Universal Robots PolyScope program: MAIN_bak20230705.urp

Program MAIN_bak20230705 (installation=GD directory=/programs/GD createdIn=5.13.0 lastSavedIn=5.13.0 robotSerialNumber=20205000017)
Calibrated DH parameters: a=[-0.000157, -0.56303, -0.236706, -0.000074, -0.000109, 0]; d=[0.181705, 47.632387, 369.599619, -417.058513, 0.119878, 0.115667]; alpha=[1.570881, -0.005074, -0.001247, 1.56886, -1.570997, 0]; deltaTheta=[0, -0.405485, 5.544791, 1.143886, -0.000009, -0.000001]
InitVariablesNode
BeforeStart
  Script file /programs/GD/ROVI/ROVI_RESET.script
    | def ROVI_RESET():
    |   if (not socket_open(host,port,socket_name)):
    |     rovi_err=902
    |     return False
    |   end
    |   socket_send_line("X0()",socket_name)
    |   ret=socket_read_line(socket_name,socket_timeout)
    |   if (ret == "OK"):
    |     rovi_err=0
    |   elif (ret == "NG"):
    |     rovi_err=to_num(socket_read_line(socket_name,socket_timeout))
    |   else:
    |     ret="NG"
    |     rovi_err=903
    |   end
    |   socket_close(socket_name)
    |   if (rovi_err != 0):
    |     if (is_popup):
    |       popup(str_cat(ret,rovi_err),title="X0",warning=True,blocking=True)
    |     end
    |     return False
    |   else:
    |     return True
    |   end
    | end
  Script file /programs/GD/ROVI/ROVI_CAPTURE.script
    | def ROVI_CAPTURE():
    |   Y1=[0.0,0.0,0.0,0.0]
    | #  p=get_actual_tool_flange_pose()
    |   p=Bucket
    |   if (not socket_open(host,port,socket_name)):
    |     rovi_err=902
    |     return False
    |   end
    |   socket_send_string("X1(",socket_name)
    |   socket_send_string(p[0],socket_name)
    |   socket_send_string(",",socket_name)
    |   socket_send_string(p[1],socket_name)
    |   socket_send_string(",",socket_name)
    |   socket_send_string(p[2],socket_name)
    |   socket_send_string(",",socket_name)
    |   socket_send_string(p[3],socket_name)
    |   socket_send_string(",",socket_name)
    |   socket_send_string(p[4],socket_name)
    |   socket_send_string(",",socket_name)
    |   socket_send_string(p[5],socket_name)
    |   socket_send_line(")",socket_name)
    |   ret=socket_read_line(socket_name,socket_timeout)
    |   if (ret == "OK"):
    |     rovi_err=0
    |     f=socket_read_ascii_float(4,socket_name,socket_timeout)
    |     while (f[0]!=4):
    |       sleep(0.3)
    |       f=socket_read_ascii_float(4,socket_name,socket_timeout)
    |     end
    |     i=0
    |     while (i<4):
    |       Y1[i]=f[i+1]
    |       i=i+1
    |     end
    |   elif (ret == "NG"):
    |     rovi_err=to_num(socket_read_line(socket_name,socket_timeout))
    |   else:
    |     ret="NG"
    |     rovi_err=903
    |   end
    |   socket_close(socket_name)
    |   if (rovi_err != 0):
    |     if (is_popup):
    |       popup(str_cat(ret,rovi_err),title="X1",warning=True,blocking=True)
    |     end
    |     return False
    |   else:
    |     return True
    |   end
    | end
  Script file /programs/GD/ROVI/ROVI_SOLVE.script
    | def ROVI_SOLVE(is_popup=is_popup):
    |   buf=p[10000.0,0.0,0.0,0.0,0.0,0.0]
    |   if (not socket_open(host,port,socket_name)):
    |     rovi_err=902
    |     return False
    |   end
    |   socket_send_line("X2()",socket_name)
    |   ret=socket_read_line(socket_name,socket_timeout)
    |   if (ret == "OK"):
    |     rovi_err=0
    |     f=socket_read_ascii_float(6,socket_name,socket_timeout)
    |     while (f[0]!=6):
    |       sleep(0.3)
    |       f=socket_read_ascii_float(6,socket_name,socket_timeout)
    |     end
    |     counter=0
    |     while (counter<6):
    |       buf[counter]=f[counter+1]
    |       counter=counter+1
    |     end
    |   elif (ret == "NG"):
    |     rovi_err=to_num(socket_read_line(socket_name,socket_timeout))
    |   else:
    |     ret="NG"
    |     rovi_err=903
    |   end
    |   sleep(1.0)
    |   socket_close(socket_name)
    |   if (rovi_err != 0):
    |     if (is_popup):
    |       popup(str_cat(ret,rovi_err),title="X2",warning=True,blocking=True)
    |     end
    |   end
    |   return buf
    | end
  Script file /programs/GD/ROVI/ROVI_RECIPE.script
    | def ROVI_RECIPE(recipe):
    |   if (not socket_open(host,port,socket_name)):
    |     rovi_err=902
    |     return False
    |   end
    |   socket_send_line(str_cat(str_cat("X3(",recipe),")"),socket_name)
    |   ret=socket_read_line(socket_name,socket_timeout)
    |   if (ret == "OK"):
    |     rovi_err=0
    |   elif (ret == "NG"):
    |     rovi_err=to_num(socket_read_line(socket_name,socket_timeout))
    |   else:
    |     ret="NG"
    |     rovi_err=903
    |   end
    |   socket_close(socket_name)
    |   if (rovi_err != 0):
    |     if (is_popup):
    |       popup(str_cat(ret,rovi_err),title="X3",warning=True,blocking=True)
    |     end
    |     return False
    |   else:
    |     return True
    |   end
    | end
  Script file /programs/GD/ROVI/ROVI_PARAM.script
    | def ROVI_PARAM(prm_name,prm_value=None):
    |   Y8=0.0
    |   if (not socket_open(host,port,socket_name)):
    |     rovi_err=902
    |     return False
    |   end
    |   socket_send_string("X8(",socket_name)
    |   socket_send_string(prm_name,socket_name)
    |   if (prm_value != None):
    |     socket_send_string(" ",socket_name)
    |     socket_send_string(prm_value,socket_name)
    |   end
    |   socket_send_line(")",socket_name)
    |   ret=socket_read_line(socket_name,socket_timeout)
    |   if (ret == "OK"):
    |     rovi_err=0
    |     if (prm_value == None):  # rosparam get
    |       Y8=to_num(socket_read_line(socket_name,socket_timeout))
    |     else:    # rosparam set
    |       f=1
    |     end
    |   elif (ret == "NG"):
    |     rovi_err=to_num(socket_read_line(socket_name,socket_timeout))
    |   else:
    |     ret="NG"
    |     rovi_err=903
    |   end
    |   socket_close(socket_name)
    |   if (rovi_err != 0):
    |     if (is_popup):
    |       popup(str_cat(ret,rovi_err),title="X8",warning=True,blocking=True)
    |     end
    |     return False
    |   else:
    |     return True
    |   end
    | end
  Script file /programs/GD/CONTROL/STATUS_CONTROL.script
    | def CHECK_VT_STATUS():
    |   write_output_boolean_register(8, read_input_boolean_register(64))   # GPBO_PCOK
    |   write_output_boolean_register(9, read_input_boolean_register(65))   # GPBO_YCAMOK
    |   write_output_integer_register(5, read_input_integer_register(24))   # GPIO_PayloadNo
    | end
  Script file /programs/GD/CONTROL/CYCLE_CONTROL.script
    | def GET_REG(prg_no):
    |   WorkPosNo=read_input_integer_register(4)-1                       # GPII_WorkPosNo
    |   CaptIndex[WorkPosNo]=read_input_integer_register(21)-1           # GPII_CaptColNo
    |   CaptRowNo=read_input_integer_register(20)-1        # GPII_CaptRowNo
    |   CaptStepZ=read_input_integer_register(6) / 1000.0         # GPII_CaptStepZ
    |   ReCaptNo=0
    |   if (prg_no==1203):
    |     ReCaptNo=read_input_integer_register(22)                # GPII_ReCaptNo
    |   end
    |   ReCaptZ=read_input_integer_register(7) / 1000.0         # GPII_ReCaptZ
    |   CutOffZDef=read_input_integer_register(11) / 1000.0          # GPII_CutOffZ
    |   CrankDepthFull=read_input_integer_register(10) / 1000.0   # GPII_FullDepth
    | end
    | 
    | def POSE_SUB(p, teach_frame):
    |   return pose_trans(inv(teach_frame), p)
    | end
    | 
    | def GET_BUCKET_UPPER(pos=0):
    |   if UseNewCaptPos:
    |     p=POSE_SUB(CaptPoint_C, BucketM)
    |     pX=[BKWidth/2,CaptPointL_dX,BKWidth-CaptPointR_dX]
    |     p[0]=pX[pos]
    |   else:
    |     captpos=[CaptPoint_C,CaptPoint_L,CaptPoint_R]
    |     p=captpos[pos]
    |     p=POSE_SUB(p, BucketM)
    |   end
    |   return p
    | end
    | 
    | def SET_BUCKET_DEF():
    |   BucketM=pBucketM
    |   if (WorkPosNo<0):
    |     Bucket=pBucketC
    |   else:
    |     Bucket=pBucket[WorkPosNo]
    |   end
    | end
    | 
    | def SET_BUCKET():
    |   SET_BUCKET_DEF()
    |   Bucket[2]=Bucket[2]-CaptStepZ*CaptRowNo
    | end
    | 
    | def SET_CV():
    |   CV=pCV
    | end
    | 
    | def SET_CAPT_INDEX():
    |   CaptIndexWk=CaptIndex[WorkPosNo]
    |   ReCaptZWk=0
    |   if (prg_no==1203):
    |     if   (ReCaptNo==0):
    |       if (CaptIndexWk==0):
    |         if (0<=DistPillarBak):
    |           CaptIndexWk=1
    |         else:
    |           CaptIndexWk=2
    |         end
    |         ReCaptZWk=0
    |       else:
    |         CaptIndexWk=0
    |         ReCaptZWk=0
    |       end
    |     elif (ReCaptNo==1):
    |       if (CaptIndexWk==0):
    |         CaptIndexWk=0
    |         ReCaptZWk=-ReCaptZ
    |       else:
    |         CaptIndexWk=CaptIndexWk
    |         ReCaptZWk=-ReCaptZ
    |       end
    |     else:
    |       if (CaptIndexWk==0):
    |         CaptIndexWk=0
    |         ReCaptZWk=ReCaptZ
    |       else:
    |         CaptIndexWk=CaptIndexWk
    |         ReCaptZWk=ReCaptZ
    |       end
    |     end
    |   end
    | end
    | 
    | def GET_CAPTPOS():
    |   SET_BUCKET()
    |   SET_CAPT_INDEX()
    |   if UseNewCaptPos:
    |     p=GET_BUCKET_UPPER(CaptIndexWk)
    |     p[2]=p[2]-ReCaptZWk
    |   else:
    |     captpos=[CaptPoint_C,CaptPoint_L,CaptPoint_R]
    |     p=captpos[CaptIndexWk]
    |     p[2]=p[2]-ReCaptZWk
    |     p=POSE_SUB(p, BucketM)
    |   end
    |   return p
    | end
    | 
    | def CHECK_CAPTPOS():
    |   isOK=((CaptStepZ*(read_input_integer_register(20)-1)) < (read_input_integer_register(9) / 1000.0))
    |   return isOK
    | end
    | 
    | def GET_ZSLIDE_POS(p):
    |   p[2]=p[2]-CaptStepZ*CaptRowNo
    |   return p
    | end
    | 
    | def END_CYCLE():
    |   stopl(1.2)
    |   end_force_mode()
    |   end_freedrive_mode()
    |   socket_close(socket_name)
    | end
    | 
    | def CHECK_SPEED(smax,f=[1,1,1,1,1,1]):
    |   s=TCPSpeed
    |   i=0
    |   while (i<6):
    |     if ((f[i]==1) and (smax[i]<s[i])):
    |       return False
    |     end
    |     i=i+1
    |   end
    |   return True
    | end
  Script file /programs/GD/CONTROL/ZONE_CONTROL.script
    | def GET_DIST(P1, P2):
    |   return pose_dist(P1, P2)
    | end
    | def CHECK_DIST_NEAR(P1, P2, th):
    |   return (GET_DIST(P1, P2) < th)
    | end
    | def DIST_HOME():
    |   return pose_dist(gHome_Position,CurrPos_p)
    | end
    | 
    | def CHECK_HOME():
    |   return (DIST_HOME()<ZoneDistTh)
    | end
    | 
    | def DIST_CVUpper():
    |   if (read_input_integer_register(4)==1):
    |     p=g2GD_pos1
    |   else:
    |     p=g1GD_pos1
    |   end
    |   return pose_dist(p,CurrPos_p)
    | end
    | 
    | def CHECK_CVUpper():
    |   return (DIST_CVUpper()<ZoneDistTh)
    | end
    | 
    | def CHECK_RB_POS(prg_no):
    |   ret=True
    |   if (prg_no==1001):
    |     ret=CHECK_EVAC()
    |   end
    |   if ((prg_no==1201) or (prg_no==1401) or (prg_no==1402) or (prg_no==6001) or (prg_no==6101) or (prg_no==6401) or (prg_no==6102) or (prg_no==7001)):
    |     ret=CHECK_HOME()
    |   end
    |   if ((prg_no==1002) or (prg_no==1241) or (prg_no==1261)):
    |     ret=CHECK_BKInside()
    |   end
    |   if (prg_no==1251):
    |     ret=(CHECK_HOME() or CHECK_CVUpper())
    |   end
    |   if (ret != True):
    |     SubPrgResult=801
    |     sleep(999999.0)
    |   end
    | end
    | 
    | def DIST_ORIGIN():
    |   p=CurrPos_p
    |   o=p
    |   o[0]=0.0
    |   o[1]=0.0
    |   return pose_dist(o,p)
    | end
    | 
    | def CHECK_EVAC_ORG():
    |   return (EvacRadiusTh<DIST_ORIGIN())
    | end
    | 
    | def CHECK_EVAC_X():
    |   return (EvacXTh[0]<CurrPos_p[0] and CurrPos_p[0]<EvacXTh[1])
    | end
    | 
    | def CHECK_EVAC_Y():
    |   return (EvacYTh[0]<CurrPos_p[1] and CurrPos_p[1]<EvacYTh[1])
    | end
    | 
    | def CHECK_EVAC_Z():
    |   return (EvacZTh[0]<CurrPos_p[2])
    | end
    | 
    | def CHECK_EVAC():
    |   ret=True
    |   ret=(ret and CHECK_EVAC_ORG())
    |   ret=(ret and CHECK_EVAC_X())
    |   ret=(ret and CHECK_EVAC_Y())
    |   ret=(ret and CHECK_EVAC_Z())
    |   return ret
    | end
    | 
    | def CHECK_BKInside():
    |   ret=True
    |   pos=read_input_integer_register(4)
    |   if (pos>2):
    |     ret=False
    |   else:
    |     if (not read_input_boolean_register(13+pos)):
    |       ret=False
    |       ver_3=read_input_boolean_register(13+pos)
    |     else:
    |       bk=pBucket[pos-1]
    |       if (pos==1):
    |         ret=(ret and CurrPos_p[0]>ZoneHomeX)
    |         ret=(ret and bk[1]-(BucketWidth-ZoneBucketGap)<CurrPos_p[1] and CurrPos_p[1]<bk[1]-ZoneBucketGap)
    |       elif (pos==2):
    |         ret=(ret and CurrPos_p[0]<-ZoneHomeX)
    |         ret=(ret and bk[1]+ZoneBucketGap<CurrPos_p[1] and CurrPos_p[1]<bk[1]+(BucketWidth-ZoneBucketGap))
    |       end
    |     end
    |   end
    |   return ret
    | end
    | 
    | def CHECK_CVOutside():
    |   ret=True
    |   ret=(ret and gCV_11_M[0]-Zone6ThX<CurrPos_p[0])
    |   ret=(ret and CurrPos_p[0]<gCV_11_M[0]+Zone6ThX)
    |   ret=(ret and gCV_11_M[1]-Zone6ThY<CurrPos_p[1])
    |   ret=(ret and CurrPos_p[1]<gCV_11_M[1]+Zone6ThY)
    |   return (not ret)
    | end
    | 
    | def CHECK_ZONE(no):
    |   if (no==1):
    |     return (CurrPos_p[2]>=Zone1ZTh)
    |   elif (no==2):
    |     return (CurrPos_p[0]>ZoneHomeX)
    |   elif (no==3):
    |     return (CurrPos_p[0]<-ZoneHomeX)
    |   elif (no==4):
    |     return CHECK_CVUpper()
    |   elif (no==5):
    |     return CHECK_BKInside()
    |   elif (no==6):
    |     return CHECK_CVOutside()
    |   end
    | end
  Script file /programs/GD/CONTROL/ALIGN_AXIS.script
    | def GET_NORM_VEC(p,axis=2):
    |   rot=p[0.0, 0.0, 0.0, p[3], p[4], p[5]]
    |   vec=p[0.0, 0.0, 0.0, 0.0, 0.0, 0.0]
    |   vec[axis]=1.0
    |   norm_p=pose_trans(rot,vec)
    |   return [norm_p[0], norm_p[1], norm_p[2]]
    | end
    | 
    | def GET_INNER_PRODUCT(v1,v2):
    |   return v1[0]*v2[0]+v1[1]*v2[1]+v1[2]*v2[2]
    | end
    | def GET_OUTER_PRODUCT(v1,v2):
    |   x=v1[1]*v2[2]-v1[2]*v2[1]
    |   y=v1[2]*v2[0]-v1[0]*v2[2]
    |   z=v1[0]*v2[1]-v1[1]*v2[0]
    |   return [x,y,z]
    | end
    | def GET_THETA(v1,v2):
    | #  cos=GET_INNER_PRODUCT(v1,v2) / norm(v1) / norm(v2)
    |   cos=GET_INNER_PRODUCT(v1,v2)
    |   g_cos=cos
    |   theta=norm(acos(cos))
    |   return theta
    | end
    | 
    | def GET_ALIGNED_POSE(target,feature,axis=2):
    |   feature_from_target=pose_trans(pose_inv(target),feature)
    |   g_f_from_t=feature_from_target
    |   nz_feature_from_target=GET_NORM_VEC(feature_from_target,axis)
    |   g_nz_f_from_t=nz_feature_from_target
    |   nz_target_from_target=[0.0, 0.0, 0.0]
    |   nz_target_from_target[axis]=1.0
    |   g_nz_t_from_t=nz_target_from_target
    | 
    |   theta=GET_THETA(nz_feature_from_target,nz_target_from_target)
    |   g_theta=theta
    |   rot_vec_n=normalize(GET_OUTER_PRODUCT(nz_target_from_target,nz_feature_from_target))
    | 
    |   if theta>d2r(90.0):
    |     theta=theta-d2r(180.0)
    |   end
    |   rot_vec=rot_vec_n * (theta)
    |   rot_p=p[0.0,0.0,0.0,rot_vec[0],rot_vec[1],rot_vec[2]]
    |   return pose_trans(target,rot_p)
    | end
    | def GET_ALIGNED_TCP(feature,axis=2):
    |   tcp=get_actual_tcp_pose()
    |   return GET_ALIGNED_POSE(tcp,feature,axis)
    | end
  Script file /programs/GD/CONTROL/ROTATE_CONTROL.script
    | def GET_TCP_FORCE_TOOL():
    |   force_torque=get_tcp_force()
    |   force_B=p[force_torque[0], force_torque[1], force_torque[2], 0, 0, 0]
    |   torque_B=p[force_torque[3], force_torque[4], force_torque[5], 0, 0, 0]
    |   tcp=get_actual_tcp_pose()
    |   rotation_BT=p[0, 0, 0, tcp[3], tcp[4], tcp[5]]
    |   force_T=pose_trans(pose_inv(rotation_BT), force_B)
    |   torque_T=pose_trans(pose_inv(rotation_BT), torque_B)
    |   force_torque_T=p[force_T[0], force_T[1], force_T[2], torque_T[0], torque_T[1], torque_T[2]]
    |   return force_torque_T
    | end
    | 
    | def CHECK_VALUE_RZ():
    |   return True
    | end
    | 
    | def GET_FORCE_VALUE_RZ(target):
    |   PoseSub= pose_sub (CurrPos_p,target)
    |   RYSub=r2d(PoseSub[4])
    |   RZSub=r2d(PoseSub[5])
    | #  if (RYSub<RZSupRYRange[0] or RZSupRYRange[1]<RYSub):
    | #    RZSupForceVal=0.0
    | #    return RZSupForceVal
    | #  end
    |   if (RZSub<0):
    |     RZMin=RZSupDegMin[0]
    |     RZRatio=RZSupRatio[0]
    |     RZOffset=RZSupOffset[0]
    |   else:
    |     RZMin=RZSupDegMin[1]
    |     RZRatio=RZSupRatio[1]
    |     RZOffset=-RZSupOffset[1]
    |   end
    |   if (norm(RZSub) >= norm(RZMin)):
    |     RZSupForceVal=(RZMin-RZSub)*RZRatio+RZOffset
    |   else:
    |     RZSupForceVal=0
    |   end
    |   if (RZSupForceVal<RZSupForceRange[0]):
    |     RZSupForceVal=RZSupForceRange[0]
    |   elif (RZSupForceRange[1]<RZSupForceVal):
    |     RZSupForceVal=RZSupForceRange[1]
    |   end
    |   if (RYSub<RZSupRYRange[0] or RZSupRYRange[1]<RYSub):
    |     RZSupForceVal=0
    |   end
    |   if ((not UseRZSupStep1) and (ForceStep==1)):
    |     RZSupForceVal=0
    |   end
    |   return RZSupForceVal
    | end
    | 
    | def GET_CVCORR_RZ(target):
    |   PoseSub=pose_sub(CurrPos_p,target)
    |   RYSub=r2d(PoseSub[4])
    |   if (RYSub<0):
    |     RYMin=-CVCorrDegMin[0]
    |     RZRatio=CVCorrRatio[0]
    |     RZOffset=-CVCorrOffset[0]
    |   else:
    |     RYMin=-CVCorrDegMin[1]
    |     RZRatio=CVCorrRatio[1]
    |     RZOffset=CVCorrOffset[1]
    |   end
    |   if (norm(RYSub) >= norm(RYMin)):
    |     CVCorrRZVal=RYSub*RZRatio+RZOffset
    |   else:
    |     CVCorrRZVal=0
    |   end
    |   return CVCorrRZVal
    | end
  SuppressedNode
    Script file /programs/GD/CONTROL/LOG.script
      | def POPUP_CAPT_OPTION():
      |   msg=""
      |   msg=str_cat(msg,str_cat(CaptIndex[WorkPosNo],","))
      |   msg=str_cat(msg,str_cat(ReCaptZ,","))
      |   msg=str_cat(msg,str_cat(prg_no,","))
      |   msg=str_cat(msg,str_cat(DistPillarBak,","))
      |   msg=str_cat(msg,str_cat(ReCaptNo,","))
      |   msg=str_cat(msg,str_cat(CaptIndexWk,","))
      |   msg=str_cat(msg,str_cat(ReCaptZWk,","))
      |   msg=str_cat(msg,str_cat(read_output_integer_register(2),","))
      |   msg=str_cat(msg,str_cat(WorkPosNo,","))
      |   msg=str_cat(msg,str_cat(CaptRowNo,","))
      |   popup(msg,title="CAPT_OPTION",warning=True,blocking=True)
      | end
Robot Program (runOnlyOnce=false)
  Script: position_deviation_warning(True,0.4)
  SetPayload (workpieceName=k10)
  Set NoAction tcp=TCP_1
  CutOffTCP := get_tcp_offset()
  Set ExpressionOutput pin=GPIO_PrgNo; expression=0
  Set DigitalOutput pin=GPBO_PrgBegin; digitalValue=0
  Set DigitalOutput pin=GPBO_PrgEnd; digitalValue=0
  Set DigitalOutput pin=GPBO_PrgRun; digitalValue=0
  Set DigitalOutput pin=GPBO_BKPosDone; digitalValue=0
  Set DigitalOutput pin=GPBO_BLStop; digitalValue=0
  Set DigitalOutput pin=GPBO_BLStart; digitalValue=0
  Set DigitalOutput pin=GPBO_Released; digitalValue=0
  Wait DigitalInput pin=GPBI_PrgStart; digitalValue=0
  Wait DigitalInput pin=GPBI_PrgStart; digitalValue=1
  Set ExpressionOutput pin=GPIO_PrgResult; expression=0
  prg_no := GPII_PrgNo
  If ( not GPBI_PrgStop≠ False ) (checkContinuously=true)
    Script: CHECK_RB_POS(prg_no)
    Set ExpressionOutput pin=GPIO_PrgNo; expression=prg_no
    Wait Sleep waitTime=0.1
    Set SingleDigitalPulseActionState SingleDigitalPulseActionState(hiPulseInSeconds=1, pin=GP_bool_out[4])
    SubPrgResult := 100
    If (SubPrgResult≟100) (checkContinuously=true)
      Script: GET_REG(prg_no)
      Switch expression=prg_no
        Case (caseValue=1001)
          Script: CHECK_RB_POS(prg_no)
          Set ExpressionOutput pin=GPIO_SubPrgNo; expression=001
          Call SUB_001
        Case (caseValue=1002)
          Set ExpressionOutput pin=GPIO_SubPrgNo; expression=102
          Call SUB_002
          Set ExpressionOutput pin=GPIO_SubPrgNo; expression=001
          Call SUB_001
        Case (caseValue=1201)
          Set ExpressionOutput pin=GPIO_SubPrgNo; expression=101
          Call SUB_101
          Set ExpressionOutput pin=GPIO_SubPrgNo; expression=102
          Call SUB_102
          Set ExpressionOutput pin=GPIO_SubPrgNo; expression=104
          SuppressedNode
            Call SUB_104
          SuppressedNode
            Call SUB_104RX
          SuppressedNode
            Call SUB_104RXF
          Call SUB_104RXFF
          Set ExpressionOutput pin=GPIO_SubPrgNo; expression=105
          Call SUB_105
          Set ExpressionOutput pin=GPIO_SubPrgNo; expression=106
          Call SUB_106
          Set ExpressionOutput pin=GPIO_SubPrgNo; expression=121
          Call SUB_121
          Set ExpressionOutput pin=GPIO_SubPrgNo; expression=122
          Call SUB_122
          Set ExpressionOutput pin=GPIO_SubPrgNo; expression=001
          Call SUB_001
          If (CandCnt≟1)
            SubPrgResult := 990
            Wait Sleep waitTime=999999
        Case (caseValue=1202)
          Set ExpressionOutput pin=GPIO_SubPrgNo; expression=102
          Call SUB_102
          Set ExpressionOutput pin=GPIO_SubPrgNo; expression=104
          SuppressedNode
            Set ExpressionOutput pin=GPIO_SubPrgNo; expression=104
          SuppressedNode
            Call SUB_104
          SuppressedNode
            Call SUB_104RX
          SuppressedNode
            Call SUB_104RXF
          Call SUB_104RXFF
          Set ExpressionOutput pin=GPIO_SubPrgNo; expression=105
          Call SUB_105
          Set ExpressionOutput pin=GPIO_SubPrgNo; expression=106
          Call SUB_106
          Set ExpressionOutput pin=GPIO_SubPrgNo; expression=121
          Call SUB_121
          Set ExpressionOutput pin=GPIO_SubPrgNo; expression=122
          Call SUB_122
          Set ExpressionOutput pin=GPIO_SubPrgNo; expression=001
          Call SUB_001
          If (CandCnt≟1)
            SubPrgResult := 990
            Wait Sleep waitTime=999999
        Case (caseValue=1203)
          Set ExpressionOutput pin=GPIO_SubPrgNo; expression=103
          Call SUB_103
          Set ExpressionOutput pin=GPIO_SubPrgNo; expression=104
          SuppressedNode
            Call SUB_104
          SuppressedNode
            Call SUB_104RX
          SuppressedNode
            Call SUB_104RXF
          Call SUB_104RXFF
          Set ExpressionOutput pin=GPIO_SubPrgNo; expression=105
          Call SUB_105
          Set ExpressionOutput pin=GPIO_SubPrgNo; expression=106
          Call SUB_106
          Set ExpressionOutput pin=GPIO_SubPrgNo; expression=121
          Call SUB_121
          Set ExpressionOutput pin=GPIO_SubPrgNo; expression=122
          Call SUB_122
          Set ExpressionOutput pin=GPIO_SubPrgNo; expression=001
          Call SUB_001
          If (CandCnt≟1)
            SubPrgResult := 990
            Wait Sleep waitTime=999999
        Case (caseValue=1241)
          Set ExpressionOutput pin=GPIO_SubPrgNo; expression=106
          Call SUB_106
          Set ExpressionOutput pin=GPIO_SubPrgNo; expression=121
          Call SUB_121
          Set ExpressionOutput pin=GPIO_SubPrgNo; expression=122
          Call SUB_122
          Set ExpressionOutput pin=GPIO_SubPrgNo; expression=001
          Call SUB_001
        Case (caseValue=1251)
          Set ExpressionOutput pin=GPIO_SubPrgNo; expression=120
          Call SUB_120
          Set ExpressionOutput pin=GPIO_SubPrgNo; expression=121
          Call SUB_121
          Set ExpressionOutput pin=GPIO_SubPrgNo; expression=122
          Call SUB_122
          Set ExpressionOutput pin=GPIO_SubPrgNo; expression=001
          Call SUB_001
        Case (caseValue=1261)
          Set ExpressionOutput pin=GPIO_SubPrgNo; expression=161
          Call SUB_161
          Set ExpressionOutput pin=GPIO_SubPrgNo; expression=001
          Call SUB_001
        Case (caseValue=1281)
          Set ExpressionOutput pin=GPIO_SubPrgNo; expression=181
          Call SUB_181
          Set ExpressionOutput pin=GPIO_SubPrgNo; expression=001
          Call SUB_001
        Case (caseValue=1401)
          Set ExpressionOutput pin=GPIO_SubPrgNo; expression=141
          Call SUB_141
          Script: pBucket[WorkPosNo]=Y2
          Set ExpressionOutput pin=GPIO_SubPrgNo; expression=143
          Call SUB_143
          Set SingleDigitalPulseActionState SingleDigitalPulseActionState(hiPulseInSeconds=1, pin=GP_bool_out[13])
        Case (caseValue=1402)
          Set ExpressionOutput pin=GPIO_SubPrgNo; expression=142
          Call SUB_142
          Set ExpressionOutput pin=GPIO_SubPrgNo; expression=001
          Call SUB_001
          Script: pCV=Y2
        Case (caseValue=3100)
          Set ExpressionOutput pin=GPIO_SubPrgNo; expression=3100
          Call SUB_3100
        Case (caseValue=6001)
          Set ExpressionOutput pin=GPIO_SubPrgNo; expression=6001
          Call SUB_6001
        Case (caseValue=6101)
          CheckMST := 0
          Set ExpressionOutput pin=GPIO_SubPrgNo; expression=6101
          Call SUB_6101
        Case (caseValue=6102)
          If (GPII_CheckMST>0)
            CheckMST := GPII_CheckMST
            WorkPosNo := -1
            CaptRowNo := 5
            SuppressedNode
              CaptRowNo := 3
            Script: SET_BUCKET()
            Set ExpressionOutput pin=GPIO_SubPrgNo; expression=6101
            Call SUB_6101
          Set ExpressionOutput pin=GPIO_SubPrgNo; expression=6102
          SuppressedNode
            Call SUB_6102
          SuppressedNode
            Call SUB_6102RX
          SuppressedNode
            Call SUB_6102RXF
          Call SUB_6102RXFF
        Case (caseValue=6401)
          Set ExpressionOutput pin=GPIO_SubPrgNo; expression=141
          Call SUB_141
          Script: pBucketM=Y2
          Script: pBucket[WorkPosNo]=Y2
        Case (caseValue=6402)
          Set ExpressionOutput pin=GPIO_SubPrgNo; expression=142
          Call SUB_6402
        Case (caseValue=7001)
          Set ExpressionOutput pin=GPIO_SubPrgNo; expression=7001
          Call SUB_7001
        Case (caseValue=7002)
          Set ExpressionOutput pin=GPIO_SubPrgNo; expression=7002
          Call SUB_7002
    Set ExpressionOutput pin=GPIO_PrgResult; expression=SubPrgResult
  Script: END_CYCLE()
  If GPBI_PrgStop≟ True
    SubPrgResult := 800
    Set ExpressionOutput pin=GPIO_PrgResult; expression=SubPrgResult
    Set ExpressionOutput pin=GPBO_PrgRun; expression=False
  Wait Sleep waitTime=0.1
  prg_no := 0
  SetPayload (workpieceName=k10)
  Set NoAction tcp=TCP_1
  If (GPIO_PrgNo≠0)
    Set SingleDigitalPulseActionState SingleDigitalPulseActionState(hiPulseInSeconds=1, pin=GP_bool_out[5])
    Set ExpressionOutput pin=GPIO_PrgNo; expression=0
  Wait DigitalInput pin=GPBI_PrgStart; digitalValue=0
  Wait DigitalInput pin=GPBI_PrgStop; digitalValue=0
Thread スレッド_2 (runOnlyOnce=false)
  Sub3100_GPII18 := GPII_RunOption
  Script: CurrPos=get_actual_tool_flange_pose()
  Script: CurrPos_p=get_actual_tcp_pose()
  Script: Currpos_p_UF0=pose_trans(pose_inv(UF), CurrPos_p)
  TCPSpeed := get_actual_tcp_speed()
  TCPForce := get_tcp_force()
  Set ExpressionOutput pin=GPBO_RBHome; expression=CHECK_HOME()
  Set ExpressionOutput pin=GPBO_AllowGoHom; expression=CHECK_EVAC()
  Set ExpressionOutput pin=GPBO_Zone01; expression=CHECK_ZONE(1)
  Set ExpressionOutput pin=GPBO_Zone02; expression=CHECK_ZONE(2)
  Set ExpressionOutput pin=GPBO_Zone03; expression=CHECK_ZONE(3)
  Set ExpressionOutput pin=GPBO_Zone04; expression=CHECK_ZONE(4)
  Set ExpressionOutput pin=GPBO_Zone05; expression=CHECK_ZONE(5)
  Set ExpressionOutput pin=GPBO_Zone06; expression=CHECK_ZONE(6)
  Script: CHECK_VT_STATUS()
  Script: sync()
SubProgram  [hidden by the author, left out]
SubProgram  [hidden by the author, left out]
SubProgram  [hidden by the author, left out]
SubProgram  [hidden by the author, left out]
SubProgram  [hidden by the author, left out]
SuppressedNode
  SubProgram  [hidden by the author, left out]
SuppressedNode
  SubProgram  [hidden by the author, left out]
SuppressedNode
  SubProgram  [hidden by the author, left out]
SubProgram -> SUB_104RXFF
SubProgram -> SUB_105
SubProgram -> SUB_106
SubProgram -> SUB_120
SubProgram -> SUB_121
SubProgram -> SUB_122
SubProgram -> SUB_141
SubProgram  [hidden by the author, left out]
SubProgram  [hidden by the author, left out]
SubProgram  [hidden by the author, left out]
SubProgram  [hidden by the author, left out]
SubProgram  [hidden by the author, left out]
SubProgram -> SUB_6001
SubProgram -> SUB_6101
SuppressedNode
  SubProgram  [hidden by the author, left out]
SuppressedNode
  SubProgram  [hidden by the author, left out]
SuppressedNode
  SubProgram  [hidden by the author, left out]
SubProgram -> SUB_6102RXFF
SubProgram  [hidden by the author, left out]
SubProgram  [hidden by the author, left out]
SubProgram  [hidden by the author, left out]
SubProgram SUB_001 [hidden by the author, left out]
SubProgram SUB_002 [hidden by the author, left out]
SubProgram SUB_101 [hidden by the author, left out]
SubProgram SUB_102 [hidden by the author, left out]
SubProgram SUB_104 [hidden by the author, left out]
SubProgram SUB_104RX [hidden by the author, left out]
SubProgram SUB_104RXF [hidden by the author, left out]
SubProgram SUB_104RXFF (keepSynchronizedWithDisk=true) programFile=/programs/GD/SUB_104RXFF.urp
  Script: SET_BUCKET()
  Folder ROVI_CAPTURE
    If ( not ROVI_CAPTURE())
      SubPrgResult := rovi_err
      Wait Sleep waitTime=999999
    CandCnt := Y1[0]
    DistPillar := Y1[1] / 1000.0
    LevelZ := Y1[2] / 1000.0
    NeighborZ := Y1[3] / 1000.0
    If (GPII_PrgNo≠1203)
      DistPillarBak := DistPillar
    If (CandCnt<1)
      SubPrgResult := 990
      Wait Sleep waitTime=999999
  Folder ROVI_SOLVE
    If (CandCnt>0)
      Y2 := ROVI_SOLVE()
      If (Y2[0]≟10000.)
        SubPrgResult := rovi_err
        Wait Sleep waitTime=999999
  UF := Y2
  Folder PICK
    SetPayload (workpieceName=k10)
    BucketDef := pBucket[WorkPosNo]
    If (CaptIndexWk≟1)
      If ((BucketDef[2]+Sub104_TiltZTh[0]<CurrPos[2]) and (CurrPos[2]<BucketDef[2]+Sub104_TiltZTh[1]))
        If (0≤DistPillar and DistPillar≤DistPillarAPTh)
          MoveL speed 200 mm/s, acceleration 70 mm/s^2 (useActiveTCP=false) tcp=TCP_1; feature=Bucket
            Waypoint TiltL (Relative): relativeFromPosition TCP in base x=-335.02 y=-289.975 z=399.986 mm, rx=-2.1962 ry=-2.2464 rz=-0.0001 rad; joints [-125.137, -72.094, -90.48, -107.417, 89.921, 53.694] deg; TCP offset x=0 y=80 z=420 mm, rx=0 ry=0 rz=0 rad; TCP in base x=-335.069 y=-289.996 z=400.008 mm, rx=2.1521 ry=2.2 rz=-0.0901 rad; joints [-128.746, -69.644, -93.066, -103.58, 93.161, 50.22] deg; feature pose in base x=326.04 y=491.74 z=0 mm, rx=0 ry=0 rz=-1.5932 rad
        Else 
          If WorkPosNo≟0
            MoveL speed 200 mm/s, acceleration 70 mm/s^2 (useActiveTCP=false) tcp=TCP_1; feature=Bucket
              Waypoint SlideL0 (Relative): relativeFromPosition TCP in base x=6.559 y=-389.302 z=60.921 mm, rx=-0.5073 ry=3.0586 rz=-0.014 rad; joints [-67.114, -66.849, -128.346, -73.737, 92.151, 4.181] deg; TCP in base x=6.579 y=-439.267 z=60.918 mm, rx=-0.5073 ry=3.0586 rz=-0.0139 rad; joints [-69.434, -72.805, -124.655, -71.563, 92.167, 1.857] deg
          Else 
            MoveL speed 200 mm/s, acceleration 70 mm/s^2 (useActiveTCP=false) tcp=TCP_1; feature=Bucket
              Waypoint SlideL1 (Relative): relativeFromPosition TCP in base x=-4.128 y=-329.518 z=106.532 mm, rx=-0.0229 ry=-3.1387 rz=-0.0019 rad; joints [-65.843, -58.986, -127.487, -83.647, 89.896, 25.103] deg; TCP in base x=-4.138 y=-279.531 z=106.538 mm, rx=-0.0228 ry=-3.1387 rz=-0.0019 rad; joints [-62.192, -52.298, -130.125, -87.703, 89.931, 28.744] deg
    ElseIf (CaptIndexWk≟2)
      If ((BucketDef[2]+Sub104_TiltZTh[0]<CurrPos[2]) and (CurrPos[2]<BucketDef[2]+Sub104_TiltZTh[1]))
        If (-DistPillarAPTh≤DistPillar and DistPillar≤0)
          MoveL speed 200 mm/s, acceleration 70 mm/s^2 (useActiveTCP=false) tcp=TCP_1; feature=Bucket
            Waypoint TiltR (Relative): relativeFromPosition TCP in base x=-335.043 y=289.982 z=399.99 mm, rx=-2.1963 ry=-2.2462 rz=0.0001 rad; joints [-194.945, -71.897, -90.609, -107.481, 89.926, -16.106] deg; TCP in base x=-335.051 y=289.972 z=400.009 mm, rx=-2.152 ry=-2.1999 rz=-0.0898 rad; joints [-189.439, -69.266, -92.671, -107.022, 85.13, -10.62] deg
        Else 
          If WorkPosNo≟0
            MoveL speed 200 mm/s, acceleration 70 mm/s^2 (useActiveTCP=false) tcp=TCP_1; feature=Bucket
              Waypoint SlideR0 (Relative): relativeFromPosition TCP in base x=6.531 y=-439.223 z=60.88 mm, rx=-0.5073 ry=3.0587 rz=-0.0137 rad; joints [-69.436, -72.808, -124.656, -71.567, 92.166, 1.857] deg; TCP in base x=6.589 y=-389.288 z=60.942 mm, rx=-0.5074 ry=3.0586 rz=-0.014 rad; joints [-67.112, -66.85, -128.343, -73.741, 92.153, 4.181] deg
          Else 
            MoveL speed 200 mm/s, acceleration 70 mm/s^2 (useActiveTCP=false) tcp=TCP_1; feature=Bucket
              Waypoint SlideR1 (Relative): relativeFromPosition TCP in base x=-4.121 y=-279.485 z=106.522 mm, rx=-0.0229 ry=-3.1387 rz=-0.0021 rad; joints [-62.196, -52.302, -130.125, -87.705, 89.936, 28.743] deg; TCP in base x=-4.165 y=-329.432 z=106.437 mm, rx=-0.0229 ry=-3.1386 rz=-0.0022 rad; joints [-65.843, -58.989, -127.494, -83.649, 89.896, 25.103] deg
    If (0≤DistPillar and DistPillar≤DistPillarAPTh)
      MoveL speed 400 mm/s, acceleration 140 mm/s^2 (useActiveTCP=false) tcp=TCP_RX; feature=UF
        Waypoint Variable (Variable): variable(featureName=gGD_4_LM)
      MoveL speed 400 mm/s, acceleration 140 mm/s^2 (useActiveTCP=false) tcp=TCP_RX; feature=UF
        Waypoint Variable (Variable): variable(featureName=gGD_3_LM_RX)
        Waypoint Variable (Variable): variable(featureName=gGD_2_LM_RX)
        Set SingleDigitalPulseActionState SingleDigitalPulseActionState(hiPulseInSeconds=1, pin=GP_bool_out[14])
        Wait Sleep waitTime=0.5
        SuppressedNode
          Popup Message (haltProgram=false message=ok? inputType=Text)
      Timer (action=Reset) variable(name=tm_handin)
      Timer (action=Start) variable=tm_handin
      Set DigitalOutput pin=digital_out[1]; digitalValue=1
      Force Frame feature=Joint_6_name; selection=[1, 1, 1, 0, 0, 0]; wrench=[0, 0, 20, 0, 0, 0]; limitsForce=[0.005, 0.005, 0.04, 0.034907, 0.034907, 1.047198]; limitsMotion=[0.1, 0.1, 0.1, 0.349066, 0.349066, 0.349066]
        Wait Condition expression=((Currpos_p_UF0[1]≤(gGD_2_LM_RX[1]-HandInZ)) or (tm_handin>GPII_TMHandIn))
      Timer (action=Stop) variable=tm_handin
      Set SingleDigitalPulseActionState SingleDigitalPulseActionState(hiPulseInSeconds=1, pin=GP_bool_out[15])
      Set DigitalOutput pin=digital_out[1]; digitalValue=0
    ElseIf (-DistPillarAPTh≤DistPillar and DistPillar≤0)
      MoveL speed 400 mm/s, acceleration 70 mm/s^2 (useActiveTCP=false) tcp=TCP_RX; feature=UF
        Waypoint Variable (Variable): variable(featureName=gGD_4_RM)
      MoveL speed 400 mm/s, acceleration 70 mm/s^2 (useActiveTCP=false) tcp=TCP_RX; feature=UF
        Waypoint Variable (Variable): variable(featureName=gGD_3_RM_RX)
        Waypoint Variable (Variable): variable(featureName=gGD_2_RM_RX)
        Set SingleDigitalPulseActionState SingleDigitalPulseActionState(hiPulseInSeconds=1, pin=GP_bool_out[14])
        Wait Sleep waitTime=0.5
        SuppressedNode
          Popup Message (haltProgram=false message=ok? inputType=Text)
      Timer (action=Reset) variable=tm_handin
      Timer (action=Start) variable=tm_handin
      Set DigitalOutput pin=digital_out[1]; digitalValue=1
      Force Frame feature=Joint_6_name; selection=[1, 1, 1, 0, 0, 0]; wrench=[0, 0, 20, 0, 0, 0]; limitsForce=[0.005, 0.005, 0.04, 0.034907, 0.034907, 1.047198]; limitsMotion=[0.1, 0.1, 0.1, 0.349066, 0.349066, 0.349066]
        Wait Condition expression=((Currpos_p_UF0[1]≤(gGD_2_RM_RX[1]-HandInZ)) or (tm_handin>GPII_TMHandIn))
      Timer (action=Stop) variable=tm_handin
      Set SingleDigitalPulseActionState SingleDigitalPulseActionState(hiPulseInSeconds=1, pin=GP_bool_out[15])
      Set DigitalOutput pin=digital_out[1]; digitalValue=0
    Else 
      MoveL speed 400 mm/s, acceleration 70 mm/s^2 (useActiveTCP=false) tcp=TCP_RX; feature=UF
        Waypoint Variable (Variable): variable(featureName=gGD_3_M_RX)
        Waypoint Variable (Variable): variable(featureName=gGD_2_M_RX)
        Set SingleDigitalPulseActionState SingleDigitalPulseActionState(hiPulseInSeconds=1, pin=GP_bool_out[14])
        Wait Sleep waitTime=0.5
        SuppressedNode
          Popup Message (haltProgram=false message=ok? inputType=Text)
      Timer (action=Reset) variable=tm_handin
      Timer (action=Start) variable=tm_handin
      Set DigitalOutput pin=digital_out[1]; digitalValue=1
      Force Frame feature=Joint_6_name; selection=[1, 1, 1, 0, 0, 0]; wrench=[0, 0, 20, 0, 0, 0]; limitsForce=[0.005, 0.005, 0.04, 0.034907, 0.034907, 1.047198]; limitsMotion=[0.1, 0.1, 0.1, 0.349066, 0.349066, 0.349066]
        ShakeCnt := -1
        Loop While (checkContinuously=false) expression=((Currpos_p_UF0[1]>(gGD_2_M_RX[1]-HandInZ)) and (tm_handin<GPII_TMHandIn))
          If UseShake
            If ShakeCnt<0
              Folder NOT_SHAKE
                Timer (action=Start) variable(name=tm_104)
                Wait Condition expression=tm_104>ShakeWaitSec
                Timer (action=Stop) variable=tm_104
                Timer (action=Reset) variable=tm_104
              ShakeCnt := 0
            IsShake := False
            Folder MONITOR_SPEED
              Timer (action=Reset) variable=tm_104
              If norm(TCPSpeed[1])<TCPSpeedThZ
                IsShake := True
                If ShakeCnt≟0
                  Timer (action=Start) variable=tm_104
                  Loop While (checkContinuously=false) expression=((tm_104<1.0) and (IsShake≟ True ))
                    If norm(TCPSpeed[1])≥TCPSpeedThZ
                      IsShake := False
                  Timer (action=Stop) variable=tm_104
                ShakeCnt := ShakeCnt+1
            Folder SHAKE
              If IsShake
                Sub3100_Option := 7
                Loop Counting (count=2) loopVariable(name=ループ_8)
                  '7:RX+,8:RX-,9:RY+,10:RY-,11:RZ+,12:RZ-'
                  Sub3100_Xd := [0.,0.,0.,0.,0.,0.]
                  Sub3100_q := floor((Sub3100_Option-1) / 2)
                  Sub3100_e := 1-((Sub3100_Option-1) % 2)*2
                  Sub3100_t := 0.2
                  Script: Sub3100_Xd[Sub3100_q]=d2r(Sub3100_XdRot/2.0)*Sub3100_e
                  Script: speedl(Sub3100_Xd,Sub3100_aRot/2.0,Sub3100_t)
                  If Sub3100_Option≟7
                    Sub3100_Option := 8
                  Else 
                    Sub3100_Option := 7
                  Wait Sleep waitTime=0.1
                IsShake := False
          Wait Sleep waitTime=0.1
      Set DigitalOutput pin=digital_out[1]; digitalValue=0
      Timer (action=Stop) variable=tm_handin
      Set SingleDigitalPulseActionState SingleDigitalPulseActionState(hiPulseInSeconds=1, pin=GP_bool_out[15])
      SuppressedNode
        IsSteady_01 := is_steady()
      SuppressedNode
        Wait Sleep waitTime=2
      SuppressedNode
        IsSteady_02 := is_steady()
    Timer (action=Reset) variable(name=tm_steady_104)
    Timer (action=Start) variable=tm_steady_104
    Wait Condition expression=is_steady()
    Timer (action=Stop) variable=tm_steady_104
    SuppressedNode
      Popup Message (haltProgram=false message=force done! inputType=Text)
    If ( not GPBI_WorkExists)
      If (0≤DistPillar and DistPillar≤DistPillarAPTh)
        MoveL speed 400 mm/s, acceleration 140 mm/s^2 (useActiveTCP=false) tcp=TCP_RX; feature=UF
          Waypoint Variable (Variable): variable(featureName=gGD_2_LM_RX)
          Waypoint Variable (Variable): variable(featureName=gGD_3_LM_RX)
        MoveL speed 400 mm/s, acceleration 140 mm/s^2 (useActiveTCP=false) tcp=TCP_RX; feature=UF
          Waypoint Variable (Variable): variable(featureName=gGD_4_LM)
      ElseIf (-DistPillarAPTh≤DistPillar and DistPillar≤0)
        MoveL speed 400 mm/s, acceleration 70 mm/s^2 (useActiveTCP=false) tcp=TCP_RX; feature=UF
          Waypoint Variable (Variable): variable(featureName=gGD_2_RM_RX)
          Waypoint Variable (Variable): variable(featureName=gGD_3_RM_RX)
        MoveL speed 400 mm/s, acceleration 70 mm/s^2 (useActiveTCP=false) tcp=TCP_RX; feature=UF
          Waypoint Variable (Variable): variable(featureName=gGD_4_RM)
      Else 
        MoveL speed 400 mm/s, acceleration 70 mm/s^2 (useActiveTCP=false) tcp=TCP_RX; feature=UF
          Waypoint Variable (Variable): variable(featureName=gGD_2_M_RX)
          Waypoint Variable (Variable): variable(featureName=gGD_3_M_RX)
      SetPayload (workpieceName=k25)
      Folder ROVI_CAPTURE
        CaptPos := GET_CAPTPOS()
        MoveL speed 400 mm/s, acceleration 140 mm/s^2 (useActiveTCP=false) tcp=TCP_1; feature=Bucket
          Waypoint Variable (Variable): variable=CaptPos
        Wait Sleep waitTime=1
        SuppressedNode
          Script: POPUP_CAPT_OPTION()
      SubPrgResult := 821
      Wait Sleep waitTime=999999
SubProgram SUB_105 (keepSynchronizedWithDisk=true) programFile=/programs/GD/SUB_105.urp
  UF := Y2
  Folder PICK
    Folder FREE_DRIVE
      SetPayload (workpieceName=k2)
      Script: freedrive_mode()
      Set NoAction tcp=ZERO
      Wait Sleep waitTime=0.5
      Script: end_freedrive_mode()
    ForceStartZ := CurrPos_p[2]
    If LevelZ<0
      CutOffZ := 0.0
    Else 
      CutOffZ := LevelZ
    CutOffZAdd := NeighborZ+BeyondZ
    SuppressedNode
      Popup Message (haltProgram=false message=zero ft_sensor... inputType=Text)
    TCPForceBak := TCPForce
    Timer (action=Reset) variable(name=tm_cutoff)
    Timer (action=Start) variable=tm_cutoff
    If (0≤DistPillar and DistPillar≤DistPillarCOTh)
      Set DigitalOutput pin=digital_out[3]; digitalValue=1
      SuppressedNode
        Force Frame feature=Bucket; selection=[1, 1, 1, 1, 1, 1]; wrench=[40, 0, 40, 0, 0, 0]; limitsForce=[0.01, 0.01, 0.015, 0.174533, 0.174533, 0.174533]; limitsMotion=[0.1, 0.1, 0.1, 0.349066, 0.349066, 0.349066]
          SetPayload (workpieceName=k05)
          CutOffZ := CutOffZ+CutOffZAdd
          Wait Condition expression=tm_cutoff>GPII_TMCutOff or CurrPos_p[2]>ForceStartZ+CutOffZ or GPBI_BLLoad2
      Folder FORCE_CUTOFF
        SetPayload (workpieceName=k1)
        Wait Sleep waitTime=0.02
        SuppressedNode
          Script: zero_ftsensor()
        ForceFeature := Bucket
        ForceValue := [40,0,40,0,0,0]
        ForceLimit := [0.01,0.01,ForceLimitZ[0],d2r(10.),d2r(10.),d2r(10.)]
        CutOffZ := CutOffZ+CutOffZAdd
        Script: force_mode(ForceFeature,ForceAxis,ForceValue,ForceType,ForceLimit)
        Loop While (checkContinuously=true) expression=tm_cutoff<GPII_TMCutOff and CurrPos_p[2]<ForceStartZ+CutOffZ and ( not GP_bool_in[11])
          If UseRZSuppress
            If WorkPosNo≟0
              Script: ForceValue[5]=-GET_FORCE_VALUE_RZ(g2GD_pos5)
            ElseIf WorkPosNo≟1
              Script: ForceValue[5]=-GET_FORCE_VALUE_RZ(g1GD_pos5)
            Script: force_mode(ForceFeature,ForceAxis,ForceValue,ForceType,ForceLimit)
          Script: sync()
        Script: end_force_mode()
        Script: stopl(1.0)
      Set DigitalOutput pin=digital_out[3]; digitalValue=0
    ElseIf (-DistPillarCOTh≤DistPillar and DistPillar≤0)
      Set DigitalOutput pin=digital_out[2]; digitalValue=1
      SuppressedNode
        Force Frame feature=Bucket; selection=[1, 1, 1, 1, 1, 1]; wrench=[-40, 0, 40, 0, 0, 0]; limitsForce=[0.01, 0.01, 0.015, 0.174533, 0.174533, 0.174533]; limitsMotion=[0.1, 0.1, 0.1, 0.349066, 0.349066, 0.349066]
          SetPayload (workpieceName=k05)
          CutOffZ := CutOffZ+CutOffZAdd
          Wait Condition expression=tm_cutoff>GPII_TMCutOff or CurrPos_p[2]>ForceStartZ+CutOffZ or GPBI_BLLoad2
      Folder FORCE_CUTOFF
        SetPayload (workpieceName=k1)
        Wait Sleep waitTime=0.02
        SuppressedNode
          Script: zero_ftsensor()
        ForceFeature := Bucket
        ForceValue := [-40,0,40,0,0,0]
        ForceLimit := [0.01,0.01,ForceLimitZ[0],d2r(10.),d2r(10.),d2r(10.)]
        CutOffZ := CutOffZ+CutOffZAdd
        Script: force_mode(ForceFeature,ForceAxis,ForceValue,ForceType,ForceLimit)
        Loop While (checkContinuously=true) expression=tm_cutoff<GPII_TMCutOff and CurrPos_p[2]<ForceStartZ+CutOffZ and ( not GP_bool_in[11])
          If UseRZSuppress
            If WorkPosNo≟0
              Script: ForceValue[5]=-GET_FORCE_VALUE_RZ(g2GD_pos5)
            ElseIf WorkPosNo≟1
              Script: ForceValue[5]=-GET_FORCE_VALUE_RZ(g1GD_pos5)
            Script: force_mode(ForceFeature,ForceAxis,ForceValue,ForceType,ForceLimit)
          Script: sync()
        Script: end_force_mode()
        Script: stopl(1.0)
      Set DigitalOutput pin=digital_out[3]; digitalValue=0
    Else 
      Set DigitalOutput pin=digital_out[3]; digitalValue=1
      SuppressedNode
        Force Frame feature=Bucket; selection=[1, 1, 1, 1, 1, 1]; wrench=[0, 0, 40, 0, 0, 0]; limitsForce=[0.01, 0.01, 0.015, 0.174533, 0.174533, 0.174533]; limitsMotion=[0.1, 0.1, 0.1, 0.349066, 0.349066, 0.349066]
          SetPayload (workpieceName=k05)
          SuppressedNode
            CutOffZ := CutOffZ+CutOffZDef
          CutOffZ := CutOffZ+CutOffZAdd
          Wait Condition expression=tm_cutoff>GPII_TMCutOff or CurrPos_p[2]>ForceStartZ+CutOffZ or GPBI_BLLoad2
      Folder FORCE_CUTOFF
        SetPayload (workpieceName=k1)
        Wait Sleep waitTime=0.02
        SuppressedNode
          Script: zero_ftsensor()
        ForceStep := 0
        ForceValue := [0,0,40,0,0,0]
        ForceFeature := Bucket
        CutOffZ := CutOffZ+CutOffZAdd
        Loop While (checkContinuously=false) expression=tm_cutoff<GPII_TMCutOff
          If WorkPosNo≟0
            Script: ForceValue[5]=-GET_FORCE_VALUE_RZ(g2GD_pos5)
          ElseIf WorkPosNo≟1
            Script: ForceValue[5]=-GET_FORCE_VALUE_RZ(g1GD_pos5)
          Switch expression=ForceStep
            Case (caseValue=0)
              ForceStep := 1
              ForceLimit := [0.01,0.01,ForceLimitZ[ForceStep-1],d2r(10.),d2r(10.),d2r(10.)]
              Script: force_mode(ForceFeature,ForceAxis,ForceValue,ForceType,ForceLimit)
            Case (caseValue=1)
              If GPBI_BLLoad1
                ForceStep := 2
                ForceLimit := [0.01,0.01,ForceLimitZ[ForceStep-1],d2r(10.),d2r(10.),d2r(10.)]
                Script: force_mode(ForceFeature,ForceAxis,ForceValue,ForceType,ForceLimit)
              ElseIf UseRZSuppress
                Script: force_mode(ForceFeature,ForceAxis,ForceValue,ForceType,ForceLimit)
            Case (caseValue=2)
              If GP_bool_in[11]
                Script: break
              If CurrPos_p[2]>ForceStartZ+CutOffZ
                ForceStep := 3
                Script: ForceValue[2]=0.0
                ForceLimit := [0.01,0.01,ForceLimitZ[ForceStep-1],d2r(10.),d2r(10.),d2r(10.)]
                Script: force_mode(ForceFeature,ForceAxis,ForceValue,ForceType,ForceLimit)
              ElseIf UseRZSuppress
                Script: force_mode(ForceFeature,ForceAxis,ForceValue,ForceType,ForceLimit)
            Case (caseValue=3)
              If GP_bool_in[11]
                Script: break
              If (UseRZSuppress and (ForceValue[5]≠0.0))
                Script: force_mode(ForceFeature,ForceAxis,ForceValue,ForceType,ForceLimit)
              Else 
                If CHECK_SPEED(StopSpeed) and ((UseRZSuppress and (ForceValue[5]==0.0)) or ( not UseRZSuppress))
                  Script: break
            SuppressedNode
              Case (caseValue=4)
                var_9 := var_9+1
                If CHECK_SPEED(StopSpeed)
                  Script: break
          Script: sync()
        Script: end_force_mode()
        Script: stopl(5.0)
      Set DigitalOutput pin=digital_out[3]; digitalValue=0
    SuppressedNode
      Wait NoWait
    SuppressedNode
      Script: end_force_mode()
    SuppressedNode
      Script: stopl(1.0)
    Set DigitalOutput pin=digital_out[3]; digitalValue=0
    Wait Condition expression=is_steady()
    Timer (action=Stop) variable=tm_cutoff
  If (GPBI_BLLoad2)
    SubPrgResult := 825
    Wait Sleep waitTime=999999
  If ( not GPBI_BLLoad1)
    SubPrgResult := 822
    Wait Sleep waitTime=999999
  SetPayload (workpieceName=k10)
  SuppressedNode
    IsSteady_01 := is_steady()
  SuppressedNode
    Wait Sleep waitTime=1.5
  SuppressedNode
    IsSteady_02 := is_steady()
  Timer (action=Reset) variable(name=tm_steady_105)
  Timer (action=Start) variable=tm_steady_105
  Wait Condition expression=is_steady()
  Timer (action=Stop) variable=tm_steady_105
  Set DigitalOutput pin=digital_out[0]; digitalValue=1
  Folder FREE_DRIVE
    Script: freedrive_mode()
    SetPayload (workpieceName=k2)
    Set NoAction tcp=ZERO
    Wait Sleep waitTime=1.5
    Script: end_freedrive_mode()
  Wait Condition expression=is_steady()
  Set DigitalOutput pin=digital_out[0]; digitalValue=0
  Folder CV_CORR_RZ
    If UseCVCorr
      Set NoAction tcp=TCP_1
      Script: sync()
      Script: CurrPos_p=get_actual_tcp_pose()
      CurrposAligned := p[0,0,0,0,0,0]
      CurrposAligned := GET_ALIGNED_TCP(CurrposAligned)
      CVCorrRZVal := GET_CVCORR_RZ(CurrposAligned)
  Folder CUTOFF_POSE
    If UseCutOffTCP
      Set NoAction tcp=TCP_1
      CutOffPos := p[0.,0.,0.,0.,0.,0.]
      CutOffPos := GET_ALIGNED_TCP(CutOffPos)
      CutOffTCP := pose_trans(pose_inv(CurrPos),CutOffPos)
      Set NoAction tcp=ZERO
      CutOffTCP := pose_trans(get_tcp_offset(),CutOffTCP)
      Set NoAction tcp=TCP_1
    Else 
      Set NoAction tcp=TCP_1
      CutOffTCP := get_tcp_offset()
SubProgram SUB_106 (keepSynchronizedWithDisk=true) programFile=/programs/GD/SUB_106.urp
  If GPBI_WorkExists (checkContinuously=true)
    Folder TRANSFER
      If (WorkPosNo≟0)
        Set DigitalOutput pin=digital_out[7]; digitalValue=1
        SetPayload (workpieceName=k120)
        If UseBaseZRotate
          Set NoAction tcp=TCP_COG
          Script: sync()
          Script: CurrPos_p=get_actual_tcp_pose()
          MoveL speed 60 mm/s, acceleration 10 mm/s^2 (useActiveTCP=false) tcp=TCP_COG; feature=Base
            PoseSub := pose_sub(CurrPos_p,g2GD_pos5_NEAR)
            RZSub := r2d(PoseSub[5])
            If (norm(PoseSub[5])≥d2r(RZTh))
              PoseAdd := pose_add(p[0,0,0,0,0,d2r(RZSub)],p[0,0,0,CurrPos_p[3],CurrPos_p[4],CurrPos_p[5]])
              PoseAdd := p[CurrPos_p[0],CurrPos_p[1],CurrPos_p[2],PoseAdd[3],PoseAdd[4],PoseAdd[5]]
              Waypoint Variable (Variable): variable=PoseAdd
        Else 
          MoveL speed 60 mm/s, acceleration 10 mm/s^2 (useActiveTCP=false) tcp=ZERO; feature=Base
            PoseSub := pose_sub(CurrPos, pose_trans(g2GD_pos5, pose_inv(get_tcp_offset())))
            RZSub := r2d(PoseSub[5])
            If (norm(PoseSub[5])≥d2r(RZTh))
              Script: PoseSub[0]=0.0
              Script: PoseSub[1]=0.0
              Script: PoseSub[2]=0.0
              PoseAdd := pose_add(PoseSub, CurrPos)
              Waypoint Variable (Variable): variable=PoseAdd
        SuppressedNode
          MoveL speed 250 mm/s, acceleration 50 mm/s^2 (useActiveTCP=false) tcp=TCP_1; feature=Base
            Waypoint Variable (Variable): variable(featureName=g2GD_pos5)
        Script: set_tcp(CutOffTCP)
        MoveL speed 250 mm/s, acceleration 50 mm/s^2 (useActiveTCP=true) feature=Base
          If UseZSlide
            gGD_pos5 := GET_ZSLIDE_POS(g2GD_pos5_NEAR)
          Else 
            gGD_pos5 := g2GD_pos5
          Script: DistBKUpper=GET_DIST(CurrPos_p,gGD_pos5)
          If ( not CHECK_DIST_NEAR(CurrPos_p, gGD_pos5, DistBKUpperTh))
            Waypoint Variable (Variable): variable=gGD_pos5
          Set DigitalOutput pin=digital_out[7]; digitalValue=0
        Set DigitalOutput pin=digital_out[6]; digitalValue=1
        MoveL speed 400 mm/s, acceleration 140 mm/s^2 (useActiveTCP=true) feature=Base
          SetPayload (workpieceName=k10)
          Waypoint Variable (Variable): variable(featureName=g2GD_pos4)
          Waypoint Variable (Variable): motionParameters(blendRadius=0.1); variable(featureName=g2GD_pos3)
          Waypoint Variable (Variable): motionParameters(jointSpeed=1.047198 jointAcceleration=1.396263 cartesianSpeed=0.4 cartesianAcceleration=0.07); variable(featureName=g2GD_pos2)
        Set DigitalOutput pin=digital_out[6]; digitalValue=0
        Set DigitalOutput pin=digital_out[4]; digitalValue=1
        MoveL speed 400 mm/s, acceleration 70 mm/s^2 (useActiveTCP=true) feature=Base
          SetPayload (workpieceName=k120)
          Waypoint Variable (Variable): motionParameters(blendRadius=0.05); variable(featureName=g2GD_pos1)
      ElseIf (WorkPosNo≟1)
        SetPayload (workpieceName=k120)
        Set NoAction tcp=TCP_COG
        If UseBaseZRotate
          Script: sync()
          Script: CurrPos_p=get_actual_tcp_pose()
          MoveL speed 60 mm/s, acceleration 10 mm/s^2 (useActiveTCP=false) tcp=TCP_COG; feature=Base
            PoseSub := pose_sub(CurrPos_p,g1GD_pos5_NEAR)
            RZSub := r2d(PoseSub[5])
            If (norm(PoseSub[5])≥d2r(RZTh))
              PoseAdd := pose_add(p[0,0,0,0,0,d2r(RZSub)],p[0,0,0,CurrPos_p[3],CurrPos_p[4],CurrPos_p[5]])
              PoseAdd := p[CurrPos_p[0],CurrPos_p[1],CurrPos_p[2],PoseAdd[3],PoseAdd[4],PoseAdd[5]]
              Waypoint Variable (Variable): variable=PoseAdd
        Else 
          MoveL speed 60 mm/s, acceleration 10 mm/s^2 (useActiveTCP=false) tcp=ZERO; feature=Base
            PoseSub := pose_sub(CurrPos, pose_trans(g1GD_pos5, pose_inv(get_tcp_offset())))
            RZSub := r2d(PoseSub[5])
            If (norm(PoseSub[5])≥d2r(RZTh))
              Script: PoseSub[0]=0.0
              Script: PoseSub[1]=0.0
              Script: PoseSub[2]=0.0
              PoseAdd := pose_add(PoseSub, CurrPos)
              Waypoint Variable (Variable): variable=PoseAdd
        SuppressedNode
          MoveL speed 250 mm/s, acceleration 50 mm/s^2 (useActiveTCP=false) tcp=TCP_1; feature=Base
            Waypoint Variable (Variable): variable(featureName=g1GD_pos5)
        Script: set_tcp(CutOffTCP)
        MoveL speed 250 mm/s, acceleration 50 mm/s^2 (useActiveTCP=true) feature=Base
          If UseZSlide
            gGD_pos5 := GET_ZSLIDE_POS(g1GD_pos5_NEAR)
          Else 
            gGD_pos5 := g1GD_pos5
          Script: DistBKUpper=GET_DIST(CurrPos_p,gGD_pos5)
          If ( not CHECK_DIST_NEAR(CurrPos_p, gGD_pos5, DistBKUpperTh))
            Waypoint Variable (Variable): variable=gGD_pos5
        Set DigitalOutput pin=digital_out[4]; digitalValue=0
        Set DigitalOutput pin=digital_out[6]; digitalValue=1
        MoveL speed 400 mm/s, acceleration 140 mm/s^2 (useActiveTCP=true) feature=Base
          SetPayload (workpieceName=k10)
          Waypoint Variable (Variable): variable(featureName=g1GD_pos3)
          Waypoint Variable (Variable): variable(featureName=g1GD_pos2)
        Set DigitalOutput pin=digital_out[6]; digitalValue=0
        Set DigitalOutput pin=digital_out[4]; digitalValue=1
        MoveL speed 400 mm/s, acceleration 140 mm/s^2 (useActiveTCP=true) feature=Base
          SetPayload (workpieceName=k120)
          Waypoint Variable (Variable): motionParameters(blendRadius=0.1); variable(featureName=g1GD_pos1)
  Set DigitalOutput pin=digital_out[4]; digitalValue=0
  If ( not GPBI_WorkExists)
    SubPrgResult := 820
    Wait Sleep waitTime=999999
SubProgram SUB_121 (keepSynchronizedWithDisk=true) programFile=/programs/GD/SUB_121.urp
  Script: SET_CV()
  If GPBI_WorkExists (checkContinuously=true)
    If GPBI_AllowGoCV≠ True
      SubPrgResult := 823
      Wait Sleep waitTime=999999
    SetPayload (workpieceName=k120)
    MoveL speed 500 mm/s, acceleration 70 mm/s^2 (useActiveTCP=true) feature=CV
      Waypoint Variable (Variable): variable(featureName=gCV_2_M)
    Script: set_tcp(CutOffTCP)
    MoveL speed 300 mm/s, acceleration 70 mm/s^2 (useActiveTCP=true) feature=CV
      Waypoint Variable (Variable): variable(featureName=gCV_1_M)
    Set NoAction tcp=TCP_1
    SuppressedNode
      Popup Message (haltProgram=false message=stop inputType=Text)
    Folder CV_CORR_RZ
      If UseCVCorr
        RZSub := CVCorrRZVal
        Set NoAction tcp=TCP_1
        Wait Sleep waitTime=0.02
        Script: CurrPos_p=get_actual_tcp_pose()
        MoveL speed 60 mm/s, acceleration 10 mm/s^2 (useActiveTCP=false) tcp=TCP_1; feature=Base
          PoseAdd := pose_add(p[0,0,0,0,0,d2r(-RZSub)],p[0,0,0,CurrPos_p[3],CurrPos_p[4],CurrPos_p[5]])
          PoseAdd := p[CurrPos_p[0],CurrPos_p[1],CurrPos_p[2],PoseAdd[3],PoseAdd[4],PoseAdd[5]]
          Waypoint Variable (Variable): variable=PoseAdd
  Set NoAction tcp=TCP_1
  If ( not GPBI_WorkExists)
    Script: stopl(1.2)
    SubPrgResult := 820
    Wait Sleep waitTime=999999
SubProgram SUB_122 (keepSynchronizedWithDisk=true) programFile=/programs/GD/SUB_122.urp
  Script: SET_CV()
  Set SingleDigitalPulseActionState SingleDigitalPulseActionState(hiPulseInSeconds=1, pin=GP_bool_out[15])
  SetPayload (workpieceName=k05)
  ForceStartZ := CurrPos[2]
  Timer (action=Reset) variable(name=tm_landed)
  Timer (action=Start) variable=tm_landed
  Set DigitalOutput pin=digital_out[5]; digitalValue=1
  Force Frame feature=CV; selection=[1, 1, 1, 0, 1, 0]; wrench=[0, 0, -40, 0, 0, 0]; limitsForce=[0.005, 0.005, 0.02, 0.174533, 0.034907, 0.174533]; limitsMotion=[0.1, 0.1, 0.1, 0.349066, 0.349066, 0.349066]
    Wait Condition expression=GPII_TMLanded<tm_landed or GPBI_BLLoad0 or CurrPos[2]<ForceStartZ-UnloadZ
    Wait Sleep waitTime=0.5
  Set DigitalOutput pin=digital_out[5]; digitalValue=0
  Script: end_force_mode()
  Timer (action=Stop) variable=tm_landed
  If ( not GPBI_BLLoad0)
    SubPrgResult := 824
    Wait Sleep waitTime=999999
  SetPayload (workpieceName=k10)
  MoveL speed 200 mm/s, acceleration 70 mm/s^2 (useActiveTCP=false) tcp=TCP_1; feature=CV
    Wait Sleep waitTime=1
    Waypoint Variable (Variable): motionParameters(jointSpeed=1.047198 jointAcceleration=1.396263 cartesianSpeed=0.03 cartesianAcceleration=0.03); variable(featureName=gCV_11_M)
    Waypoint Variable (Variable): variable(featureName=gCV_12_M)
  Set SingleDigitalPulseActionState SingleDigitalPulseActionState(hiPulseInSeconds=3, pin=GP_bool_out[17])
  MoveL speed 500 mm/s, acceleration 140 mm/s^2 (useActiveTCP=false) tcp=TCP_1; feature=CV
    Waypoint Variable (Variable): motionParameters(blendRadius=0.05); variable(featureName=gCV_13_M)
  SetPayload (workpieceName=k10)
SubProgram SUB_103 [hidden by the author, left out]
SubProgram SUB_120 (keepSynchronizedWithDisk=true) programFile=/programs/GD/SUB_120.urp
  If GPBI_WorkExists (checkContinuously=true)
    Folder TRANSFER
      Script: set_tcp(CutOffTCP)
      MoveL speed 150 mm/s, acceleration 30 mm/s^2 (useActiveTCP=true) feature=Base
        SetPayload (workpieceName=k10)
        Waypoint Variable (Variable): variable(featureName=g2GD_pos1)
        Wait Sleep waitTime=0.5
  If ( not GPBI_WorkExists)
    SubPrgResult := 820
    Wait Sleep waitTime=999999
SubProgram SUB_161 [hidden by the author, left out]
SubProgram SUB_181 [hidden by the author, left out]
SubProgram SUB_141 (keepSynchronizedWithDisk=true) programFile=/programs/GD/SUB_141.urp
  Folder INITIALIZE
    SetPayload (workpieceName=k10)
    Script: pBucket[WorkPosNo]=p[0.,0.,0.,0.,0.,0.]
    If (WorkPosNo≟0)
      GD_pos4 := Capt_2BK_pos1
      GD_pos5 := Capt_2BK_pos2
      Capt_BK_L := Capt_2BK_L
      Capt_BK_R := Capt_2BK_R
    ElseIf (WorkPosNo≟1)
      GD_pos4 := Capt_1BK_pos1
      GD_pos5 := Capt_1BK_pos2
      Capt_BK_L := Capt_1BK_L
      Capt_BK_R := Capt_1BK_R
  Folder HOME
    SuppressedNode
      MoveJ speed 70 deg/s, acceleration 30 deg/s^2 (useActiveTCP=false) tcp=TCP_1; feature=Base
        Waypoint Variable (Variable): variable(name=GD_pos4)
    SuppressedNode
      MoveL speed 200 mm/s, acceleration 70 mm/s^2 (useActiveTCP=true) feature=Base
        Waypoint Variable (Variable): variable(name=GD_pos5)
  Folder ROVI_RECIPE
    If ( not ROVI_RECIPE(GPII_BucketNo))
      SubPrgResult := rovi_err
      Wait Sleep waitTime=999999
  Folder ROVI_RESET
    If ( not ROVI_RESET())
      SubPrgResult := rovi_err
      Wait Sleep waitTime=999999
  Folder ROVI_CAPTURE_1
    MoveL speed 250 mm/s, acceleration 140 mm/s^2 (useActiveTCP=false) tcp=TCP_1; feature=Base
      Waypoint Variable (Variable): variable(name=Capt_BK_L)
    Wait Sleep waitTime=1
    If ( not ROVI_CAPTURE())
      SubPrgResult := rovi_err
      Wait Sleep waitTime=999999
  Folder ROVI_CAPTURE_2
    MoveL speed 500 mm/s, acceleration 140 mm/s^2 (useActiveTCP=false) tcp=TCP_1; feature=Base
      Waypoint Variable (Variable): variable(name=Capt_BK_R)
    Wait Sleep waitTime=1
    If ( not ROVI_CAPTURE())
      SubPrgResult := rovi_err
      Wait Sleep waitTime=999999
  Folder ROVI_SOLVE
    Y2 := ROVI_SOLVE()
    If (Y2[0]≟10000.)
      SubPrgResult := rovi_err
      Wait Sleep waitTime=999999
  Folder ROVI_PARAM
    If not ROVI_PARAM(BKWidth_Name)
      SubPrgResult := rovi_err
      Wait Sleep waitTime=999999
    Script: BKWidth_Value[WorkPosNo]=Y8
  Folder HOME
    SuppressedNode
      MoveL speed 250 mm/s, acceleration 140 mm/s^2 (useActiveTCP=false) tcp=TCP_1; feature=Base
        Waypoint Variable (Variable): variable=GD_pos5
        Waypoint Variable (Variable): variable=GD_pos4
SubProgram SUB_143 [hidden by the author, left out]
SubProgram SUB_142 [hidden by the author, left out]
SubProgram SUB_3100 [hidden by the author, left out]
SubProgram SUB_6001 (keepSynchronizedWithDisk=true) programFile=/programs/GD/SUB_6001.urp
  SetPayload (workpieceName=k10)
  If ( not ROVI_RESET())
    SubPrgResult := rovi_err
    Wait Sleep waitTime=999999
  MoveJ speed 9 deg/s, acceleration 15 deg/s^2 (useActiveTCP=false) tcp=ZERO; feature=Base
    Waypoint CaptPos0: TCP in base x=62.941 y=-648.805 z=499.602 mm, rx=-0.058 ry=3.1227 rz=0.0129 rad; joints [-69.438, -86.827, -111.279, -71.978, 91.038, 18.526] deg
  CaptPos := CaptPos0_p
  Loop While (checkContinuously=false) expression=(CaptPos[0]≠10000.0)
    MoveJ speed 9 deg/s, acceleration 15 deg/s^2 (useActiveTCP=false) tcp=ZERO; feature=Base
      Waypoint Variable (Variable): variable=CaptPos
    Wait Sleep waitTime=4
    If ( not ROVI_CAPTURE())
      SubPrgResult := rovi_err
      Wait Sleep waitTime=999999
    CaptPos := ROVI_SOLVE(is_popup=False)
  MoveJ speed 9 deg/s, acceleration 15 deg/s^2 (useActiveTCP=false) tcp=ZERO; feature=Base
    Waypoint CaptPos0: TCP in base x=62.941 y=-648.805 z=499.602 mm, rx=-0.058 ry=3.1227 rz=0.0129 rad; joints [-69.438, -86.827, -111.279, -71.978, 91.038, 18.526] deg
SubProgram SUB_6101 (keepSynchronizedWithDisk=true) programFile=/programs/GD/SUB_6101.urp
  Folder ROVI_RECIPE
    If (not ROVI_RECIPE(GPII_WorkNo))
      SubPrgResult := rovi_err
      Wait Sleep waitTime=999999
  Folder ROVI_RESET
    If ( not ROVI_RESET())
      SubPrgResult := rovi_err
      Wait Sleep waitTime=999999
  Folder ROVI_CAPTURE_1
    MoveJ speed 6 deg/s, acceleration 12 deg/s^2 (useActiveTCP=false) tcp=TCP_1; feature=Base
      Switch expression=CheckMST
        Case (caseValue=0)
          Waypoint Variable (Variable): variable(featureName=Master_pos)
        Case (caseValue=1)
          Waypoint Variable (Variable): variable(featureName=Master_pos)
        Case (caseValue=2)
          Waypoint Variable (Variable): variable(featureName=Master_posL)
        Case (caseValue=3)
          Waypoint Variable (Variable): variable(featureName=Master_posR)
      SuppressedNode
        Waypoint ウェイポイント_1 (Relative): relativeFromPosition TCP in base x=-5.037 y=-329.575 z=16.043 mm, rx=-0.0235 ry=-3.1385 rz=-0.002 rad; joints [-65.945, -61.292, -135.715, -73.119, 89.887, 25.023] deg; TCP offset x=0 y=80 z=420 mm, rx=0 ry=0 rz=0 rad; TCP in base x=-3.24 y=-405.091 z=93.349 mm, rx=0.0238 ry=2.9687 rz=0.0105 rad; joints [-81.058, -70.218, -123.998, -74.522, 99.793, 10.078] deg
    Wait Sleep waitTime=3
    If ( not ROVI_CAPTURE())
      SubPrgResult := rovi_err
      Wait Sleep waitTime=999999
SubProgram SUB_6102 [hidden by the author, left out]
SubProgram SUB_6102RX [hidden by the author, left out]
SubProgram SUB_6102RXF [hidden by the author, left out]
SubProgram SUB_6102RXFF (keepSynchronizedWithDisk=true) programFile=/programs/GD/SUB_6102RXFF.urp
  SetPayload (workpieceName=k10)
  UF := Base
  If (GPII_CheckMST>0)
    Folder ROVI_SOLVE
      If (CandCnt>0)
        Y2 := ROVI_SOLVE()
        If (Y2[0]≟10000.)
          SubPrgResult := rovi_err
          Wait Sleep waitTime=999999
    UF := Y2
  Folder M
    MoveL speed 120 mm/s, acceleration 70 mm/s^2 (useActiveTCP=false) tcp=TCP_RX; feature=UF
      Waypoint Variable (Variable): variable(featureName=gGD_3_M_RX)
      Wait Sleep waitTime=1
      Waypoint Variable (Variable): variable(featureName=gGD_2_M_RX)
      Wait Sleep waitTime=1
      Set SingleDigitalPulseActionState SingleDigitalPulseActionState(hiPulseInSeconds=1, pin=GP_bool_out[14])
      Popup Message (haltProgram=false message=ok? inputType=Text)
    Timer (action=Reset) variable(name=tm_6102_01)
    Timer (action=Start) variable=tm_6102_01
    Force Frame feature=Joint_6_name; selection=[1, 1, 1, 0, 0, 0]; wrench=[0, 0, 10, 0, 0, 0]; limitsForce=[0.005, 0.005, 0.04, 0.034907, 0.034907, 1.047198]; limitsMotion=[0.1, 0.1, 0.1, 0.349066, 0.349066, 0.349066]
      ShakeCnt := -1
      Loop While (checkContinuously=false) expression=((Currpos_p_UF0[1]>(gGD_2_M_RX[1]-HandInZ)) and (tm_6102_01<GPII_TMHandIn))
        IsShake := False
        If ShakeCnt<0
          Folder NOT_SHAKE
            Timer (action=Start) variable(name=tm_6102_02)
            Wait Condition expression=tm_6102_02>ShakeWaitSec
            Timer (action=Stop) variable=tm_6102_02
            Timer (action=Reset) variable=tm_6102_02
          ShakeCnt := 0
        Folder MONITOR_SPEED
          Timer (action=Reset) variable=tm_6102_02
          If norm(TCPSpeed[2])<TCPSpeedThZ
            IsShake := True
            If ShakeCnt≟0
              Timer (action=Start) variable=tm_6102_02
              Loop While (checkContinuously=false) expression=((tm_6102_02<1.0) and (IsShake≟ True ))
                If norm(TCPSpeed[2])≥TCPSpeedThZ
                  IsShake := False
              Timer (action=Stop) variable=tm_6102_02
            ShakeCnt := ShakeCnt+1
        Folder SHAKE
          If IsShake
            Sub3100_Option := 9
            Loop Counting (count=2) loopVariable(name=ループ_6)
              '7:RX+,8:RX-,9:RY+,10:RY-,11:RZ+,12:RZ-'
              Sub3100_Xd := [0.,0.,0.,0.,0.,0.]
              Sub3100_q := floor((Sub3100_Option-1) / 2)
              Sub3100_e := 1-((Sub3100_Option-1) % 2)*2
              Sub3100_t := 0.2
              Script: Sub3100_Xd[Sub3100_q]=d2r(Sub3100_XdRot/2.0)*Sub3100_e
              Script: speedl(Sub3100_Xd,Sub3100_aRot/2.0,Sub3100_t)
              If Sub3100_Option≟9
                Sub3100_Option := 10
              Else 
                Sub3100_Option := 9
              Wait Sleep waitTime=0.1
            IsShake := False
        Wait Sleep waitTime=0.1
    Timer (action=Stop) variable=tm_6102_01
    Set SingleDigitalPulseActionState SingleDigitalPulseActionState(hiPulseInSeconds=1, pin=GP_bool_out[15])
    Wait Sleep waitTime=1
    Popup Message (haltProgram=false message=ok? inputType=Text)
    MoveL speed 120 mm/s, acceleration 70 mm/s^2 (useActiveTCP=false) tcp=TCP_RX; feature=UF
      Waypoint Variable (Variable): variable(featureName=gGD_2_M_RX)
      Wait Sleep waitTime=1
      Waypoint Variable (Variable): variable(featureName=gGD_3_M_RX)
      Wait Sleep waitTime=1
  Folder LM
    MoveL speed 120 mm/s, acceleration 70 mm/s^2 (useActiveTCP=false) tcp=TCP_RX; feature=UF
      Waypoint Variable (Variable): variable(featureName=gGD_3_LM_RX)
      Wait Sleep waitTime=1
      Waypoint Variable (Variable): variable(featureName=gGD_2_LM_RX)
      Wait Sleep waitTime=1
      Set SingleDigitalPulseActionState SingleDigitalPulseActionState(hiPulseInSeconds=1, pin=GP_bool_out[14])
      Popup Message (haltProgram=false message=ok? inputType=Text)
    Timer (action=Reset) variable=tm_6102_01
    Timer (action=Start) variable=tm_6102_01
    Force Frame feature=Joint_6_name; selection=[1, 1, 1, 0, 0, 0]; wrench=[0, 0, 10, 0, 0, 0]; limitsForce=[0.005, 0.005, 0.04, 0.034907, 0.034907, 1.047198]; limitsMotion=[0.1, 0.1, 0.1, 0.349066, 0.349066, 0.349066]
      Wait Condition expression=((Currpos_p_UF0[1]≤(gGD_2_LM_RX[1]-HandInZ)) or (tm_6102_01>GPII_TMHandIn))
    Timer (action=Stop) variable=tm_6102_01
    Set SingleDigitalPulseActionState SingleDigitalPulseActionState(hiPulseInSeconds=1, pin=GP_bool_out[15])
    Wait Sleep waitTime=1
    Popup Message (haltProgram=false message=ok? inputType=Text)
    MoveL speed 120 mm/s, acceleration 70 mm/s^2 (useActiveTCP=false) tcp=TCP_RX; feature=UF
      Waypoint Variable (Variable): variable(featureName=gGD_2_LM_RX)
      Wait Sleep waitTime=1
      Waypoint Variable (Variable): variable(featureName=gGD_3_LM_RX)
      Wait Sleep waitTime=1
  Folder RM
    MoveL speed 120 mm/s, acceleration 70 mm/s^2 (useActiveTCP=false) tcp=TCP_RX; feature=UF
      Waypoint Variable (Variable): variable(featureName=gGD_3_RM_RX)
      Wait Sleep waitTime=1
      Waypoint Variable (Variable): variable(featureName=gGD_2_RM_RX)
      Wait Sleep waitTime=1
      Set SingleDigitalPulseActionState SingleDigitalPulseActionState(hiPulseInSeconds=1, pin=GP_bool_out[14])
      Popup Message (haltProgram=false message=ok? inputType=Text)
    Timer (action=Reset) variable=tm_6102_01
    Timer (action=Start) variable=tm_6102_01
    Force Frame feature=Joint_6_name; selection=[1, 1, 1, 0, 0, 0]; wrench=[0, 0, 10, 0, 0, 0]; limitsForce=[0.005, 0.005, 0.04, 0.034907, 0.034907, 1.047198]; limitsMotion=[0.1, 0.1, 0.1, 0.349066, 0.349066, 0.349066]
      Wait Condition expression=((Currpos_p_UF0[1]≤(gGD_2_RM_RX[1]-HandInZ)) or (tm_6102_01>GPII_TMHandIn))
    Timer (action=Stop) variable=tm_6102_01
    Set SingleDigitalPulseActionState SingleDigitalPulseActionState(hiPulseInSeconds=1, pin=GP_bool_out[15])
    Wait Sleep waitTime=1
    Popup Message (haltProgram=false message=ok? inputType=Text)
    MoveL speed 120 mm/s, acceleration 70 mm/s^2 (useActiveTCP=false) tcp=TCP_RX; feature=UF
      Waypoint Variable (Variable): variable(featureName=gGD_2_RM_RX)
      Wait Sleep waitTime=1
      Waypoint Variable (Variable): variable(featureName=gGD_3_RM_RX)
      Wait Sleep waitTime=1
  MoveL speed 120 mm/s, acceleration 70 mm/s^2 (useActiveTCP=false) tcp=TCP_1; feature=Base
    Waypoint Variable (Variable): variable(featureName=gHome_Position)
SubProgram SUB_6402 [hidden by the author, left out]
SubProgram SUB_7001 [hidden by the author, left out]
SubProgram SUB_7002 [hidden by the author, left out]
